TYPE TmsSwitchInfo :
STRUCT
	State : TmsSwitchState;
	Mode : TmsSwitchMode;
	Position : TmsSwitchPosition;
	ActPos : MC_LREAL;
END_STRUCT
END_TYPE

(* stored: Version 1.1.0.1, ProductVersion 3.1.4024.11
   DUT TmsSwitchInfo: Id {9213fa35-a630-498e-967e-46661586c5ec} *)
